TYPE TYP_UR_PN_TCP :
STRUCT
	Position : TYP_REAL_XYZ;
	PositionR : TYP_REAL_XYZ;
	Velocity : TYP_REAL_XYZ;
	VelocityR : TYP_REAL_XYZ;
	Force : TYP_REAL_XYZ;
	Torque : TYP_REAL_XYZ;
	ForceScalar : REAL;
END_STRUCT
END_TYPE

(* stored: Version 1.1.0.1, ProductVersion 3.1.4024.12
   DUT TYP_UR_PN_TCP: Id {80822bd5-255c-471c-94db-1bc722ab0af7} *)
